// TIA Portal V19 export
DATA_BLOCK "POST_Request_DB"   // DB8
// stored: AutoNumber false, InstanceOfName POST_Request, InstanceOfType FB
"POST_Request"
   // VAR_INPUT
   //    start : Bool;
   //    url : String;
   //    data : String;
   // END_VAR
   // VAR_OUTPUT
   //    connected : Bool;
   //    done : Bool;
   //    busy : Bool;
   //    error : Bool;
   //    status : Word;
   //    diagnostics : "typeDiagnostics";
   //    responseCode : UInt;
   //    length : UDInt;
   // END_VAR
   // VAR_IN_OUT
   //    responseData : Array[*] of Char;
   // END_VAR
   // VAR
   //    hwID : HW_ANY;
   //    connID : CONN_OUC := 16#0001;
   //    keepConnection : Bool;
   // END_VAR
BEGIN
END_DATA_BLOCK
